// TIA Portal V20 export
TYPE "typeEm7Standard"
// stored: Access Published, Namespace Unit1
   STRUCT
      commands { ExternalWritable := 'False'} : "Unit1.typeEm7Commands";
      monitoring { ExternalWritable := 'False'} : "Unit1.typeEm7Monitoring";
   END_STRUCT;
END_TYPE
